INTERFACE InterfaceObserver

METHOD subscribe_job_directory : BOOL
VAR_INPUT
	executor: I_Job; // Represent reference to subscribed job object
END_VAR
END_METHOD

METHOD subscribe_job_event : BOOL
VAR_INPUT
	subject	  : T_MaxString;	// Subject text of event
	old_state : E_FutureExecutionState; // Job state before transition.
	new_state : E_FutureExecutionState; // Job state after transition.
	record_time	: T_FILETIME64; // File-time at the time of transition.
	executor	: I_Job; // Reference to job instance of which transition occurs.
END_VAR
END_METHOD

END_INTERFACE

(* stored: Version 1.1.0.1, ProductVersion 3.1.4026.13
   Itf InterfaceObserver: Id {90b4d035-ce37-43c5-a5a2-947514da7e7e}
   Method subscribe_job_directory: Id {8f9013c8-5018-4e79-b936-7283b70651f0}
   Method subscribe_job_event: Id {09caa5d0-8b39-4577-9c48-876741e7c7cd} *)
